// TIA Portal V20 export
TYPE "type_emRelations_em5_SoftCam"
// stored: Access Published, Namespace Unit1
   STRUCT
      transferPnPLeftAxisX : Struct
         pos00_wait : "LER_typeSoftCamPosition";
         pos01_sideTape : "LER_typeSoftCamPosition";
         pos02_hotPressLeft : "LER_typeSoftCamPosition";
         pos03_hotPressRight : "LER_typeSoftCamPosition";
         pos04_hipotThickness : "LER_typeSoftCamPosition";
         pos05_posistion : "LER_typeSoftCamPosition";
         pos06_posistion : "LER_typeSoftCamPosition";
         pos07_posistion : "LER_typeSoftCamPosition";
         pos08_posistion : "LER_typeSoftCamPosition";
         pos09_sideTapeZone : "LER_typeSoftCamPosition";
         pos10_posistion : "LER_typeSoftCamPosition";
         pos11_posistion : "LER_typeSoftCamPosition";
         pos12_posistion : "LER_typeSoftCamPosition";
         pos13_posistion : "LER_typeSoftCamPosition";
         pos14_posistion : "LER_typeSoftCamPosition";
         pos15_posistion : "LER_typeSoftCamPosition";
      END_STRUCT;
      transferPnPLeftAxisY : Struct
         pos00_wait : "LER_typeSoftCamPosition";
         pos01_sideTape : "LER_typeSoftCamPosition";
         pos02_hotPressLeft : "LER_typeSoftCamPosition";
         pos03_hotPressRight : "LER_typeSoftCamPosition";
         pos04_hipotThickness : "LER_typeSoftCamPosition";
         pos05_position : "LER_typeSoftCamPosition";
         pos06_position : "LER_typeSoftCamPosition";
         pos07_position : "LER_typeSoftCamPosition";
         pos08_noInterferenceZone : "LER_typeSoftCamPosition";
         pos09_sideTapeZone : "LER_typeSoftCamPosition";
         pos10_position : "LER_typeSoftCamPosition";
         pos11_position : "LER_typeSoftCamPosition";
         pos12_position : "LER_typeSoftCamPosition";
         pos13_position : "LER_typeSoftCamPosition";
         pos14_position : "LER_typeSoftCamPosition";
         pos15_position : "LER_typeSoftCamPosition";
      END_STRUCT;
      transferPnPLeftAxisZ : Struct
         pos00_wait : "LER_typeSoftCamPosition";
         pos01_sideTape : "LER_typeSoftCamPosition";
         pos02_hotPressLeft : "LER_typeSoftCamPosition";
         pos03_hotPressRight : "LER_typeSoftCamPosition";
         pos04_hipotThickness : "LER_typeSoftCamPosition";
         pos05_posistion : "LER_typeSoftCamPosition";
         pos06_posistion : "LER_typeSoftCamPosition";
         pos07_posistion : "LER_typeSoftCamPosition";
         pos08_posistion : "LER_typeSoftCamPosition";
         pos09_posistion : "LER_typeSoftCamPosition";
         pos10_posistion : "LER_typeSoftCamPosition";
         pos11_posistion : "LER_typeSoftCamPosition";
         pos12_posistion : "LER_typeSoftCamPosition";
         pos13_posistion : "LER_typeSoftCamPosition";
         pos14_posistion : "LER_typeSoftCamPosition";
         pos15_posistion : "LER_typeSoftCamPosition";
      END_STRUCT;
      transferPnPRightAxisX : Struct
         pos00_wait : "LER_typeSoftCamPosition";
         pos01_hipotThickness : "LER_typeSoftCamPosition";
         pos02_vision : "LER_typeSoftCamPosition";
         pos03_laserMark : "LER_typeSoftCamPosition";
         pos04_weightCheck : "LER_typeSoftCamPosition";
         pos05_posistion : "LER_typeSoftCamPosition";
         pos06_posistion : "LER_typeSoftCamPosition";
         pos07_posistion : "LER_typeSoftCamPosition";
         pos08_posistion : "LER_typeSoftCamPosition";
         pos09_posistion : "LER_typeSoftCamPosition";
         pos10_posistion : "LER_typeSoftCamPosition";
         pos11_posistion : "LER_typeSoftCamPosition";
         pos12_posistion : "LER_typeSoftCamPosition";
         pos13_posistion : "LER_typeSoftCamPosition";
         pos14_posistion : "LER_typeSoftCamPosition";
         pos15_posistion : "LER_typeSoftCamPosition";
      END_STRUCT;
      transferPnPRightAxisY : Struct
         pos00_wait : "LER_typeSoftCamPosition";
         pos01_hipotThickness : "LER_typeSoftCamPosition";
         pos02_vision : "LER_typeSoftCamPosition";
         pos03_laserMark : "LER_typeSoftCamPosition";
         pos04_weightCheck : "LER_typeSoftCamPosition";
         pos05_position : "LER_typeSoftCamPosition";
         pos06_position : "LER_typeSoftCamPosition";
         pos07_position : "LER_typeSoftCamPosition";
         pos08_noInterferenceZone : "LER_typeSoftCamPosition";
         pos09_position : "LER_typeSoftCamPosition";
         pos10_position : "LER_typeSoftCamPosition";
         pos11_position : "LER_typeSoftCamPosition";
         pos12_position : "LER_typeSoftCamPosition";
         pos13_position : "LER_typeSoftCamPosition";
         pos14_position : "LER_typeSoftCamPosition";
         pos15_position : "LER_typeSoftCamPosition";
      END_STRUCT;
      transferPnPRightAxisZ : Struct
         pos00_wait : "LER_typeSoftCamPosition";
         pos01_hipotThickness : "LER_typeSoftCamPosition";
         pos02_vision : "LER_typeSoftCamPosition";
         pos03_laserMark : "LER_typeSoftCamPosition";
         pos04_weightCheck1 : "LER_typeSoftCamPosition";
         pos05_weightCheck2 : "LER_typeSoftCamPosition";
         pos06_posistion : "LER_typeSoftCamPosition";
         pos07_posistion : "LER_typeSoftCamPosition";
         pos08_posistion : "LER_typeSoftCamPosition";
         pos09_posistion : "LER_typeSoftCamPosition";
         pos10_posistion : "LER_typeSoftCamPosition";
         pos11_posistion : "LER_typeSoftCamPosition";
         pos12_posistion : "LER_typeSoftCamPosition";
         pos13_posistion : "LER_typeSoftCamPosition";
         pos14_posistion : "LER_typeSoftCamPosition";
         pos15_posistion : "LER_typeSoftCamPosition";
      END_STRUCT;
   END_STRUCT;
END_TYPE
